// TIA Portal project "md_tarikul_islam_sheam(Batch_04)_roll_25_distribution" (V18)

(* hardware
DEVICE "S7-1500/ET200MP station_1"  S7-1500 station
   slot 0: "Rail_0"  Rack  6ES7 590-1***0-0AA0
   slot 1: "PLC_1"  CPU 1516-3 PN/DP  6ES7 516-3AN02-0AB0  V2.9
      slot 3: "CPU display_1"  6ES7591-1BA00-0AA0
      slot 32768: "PROFINET interface_1"  X1
      slot 33024: "PROFINET interface_2"  X2
      slot 33280: "DP interface_1"  X3
      slot 34817: "Virtual CP interface port_1"  Virtual CP interface port  Virtual CP interface port
   slot 2: "DI 32x24VDC HF_1"  DI 32x24VDC HF  6ES7 521-1BL00-0AB0  V2.2
   slot 3: "DQ 32x24VDC/0.5A HF_1"  DQ 32x24VDC/0.5A HF  6ES7 522-1BL01-0AB0  V1.1
   slot 4: "AI 8xU/I/RTD/TC ST_1"  AI 8xU/I/RTD/TC ST  6ES7 531-7KF00-0AB0  V2.2
   slot 5: "AQ 4xU/I ST_1"  AQ 4xU/I ST  6ES7 532-5HD00-0AB0  V2.2
DEVICE "HMI_1"  TP700 Comfort
   slot 0: "HMI_1"  TP700 Comfort  6AV2 124-0GC01-0AX0  17.0.0.0
   slot 1: "HMI_RT_1"  TP700 Comfort  6AV2 124-0GC01-0AX0  17.0.0.0
   slot 5: "HMI_1.IE_CP_1"  PROFINET Interface  17.0.0.0
      slot 1: "PROFINET Interface_1"  PROFINET Interface
         slot 1: "Port_1"  Port
         slot 2: "Port_2"  Port
   slot 7: "HMI_1.MPI/DP_CP_1"  MPI/DP Interface  17.0.0.0
*)

// ===== PLC "PLC_1"  CPU 1516-3 PN/DP =====

VAR_GLOBAL   // PLC tag table "Default tag table"
   "start" AT %I1.0 : Bool;
END_VAR

VAR_GLOBAL   // PLC tag table "Tag table_1"
   "is_mag_empty" AT %I0.6 : Bool;
   "ejecter_retracted" AT %I0.4 : Bool;
   "ejector_adv" AT %I0.5 : Bool;
   "con_fwd" AT %Q0.0 : Bool;
   "cov_back" AT %Q0.1 : Bool;
   "wp_end" AT %I0.2 : Bool;
   "stop" AT %I1.1 : Bool;
   "mag_empty_led" AT %Q1.2 : Bool;
   "advanced_slide" AT %Q0.4 : Bool;
   "cyl_advance" AT %M8.0 : Bool;
   "cyl_return" AT %M7.1 : Bool;
   "conv_fwd" AT %M7.2 : Bool;
   "cov_stop" AT %M7.3 : Bool;
   "end" AT %M7.4 : Bool;
   "mag_empty_relay" AT %M7.0 : Bool;
   "emo_relay" AT %M7.5 : Bool;
   "reset" AT %I1.3 : Bool;
   "reset_relay" AT %M7.6 : Bool;
   "mem_stop" AT %M2.0 : Bool;
   "meme_start" AT %M2.3 : Bool;
   "Tag_1" AT %M2.6 : Bool;
   "PRODUCT_END" AT %M2.7 : Bool;
   "mem_start_indicator" AT %M6.0 : Bool;
   "mem_stop_indicator" AT %M6.1 : Bool;
   "start_indicator_light" AT %Q1.0 : Bool;
   "stop_indicator_light" AT %Q1.3 : Bool;
   "reset_indicator" AT %Q1.1 : Bool;
   "mem_ready_to_go" AT %M9.0 : Bool;
   "mem_reset" AT %M3.0 : Bool;
   "mem_e_stop" AT %M3.2 : Bool;
END_VAR

ORGANIZATION_BLOCK "Main"   // OB1, LAD, ProgramCycle
TITLE = "Main Program Sweep (Cycle)"
{ S7_Optimized_Access := 'TRUE' }
VERSION : 0.1
   VAR_INPUT
      Initial_Call : Bool;   // Initial call of this OB
      Remanence : Bool;   // =True, if remanent data are available
   END_VAR
BEGIN

REGION Network 1
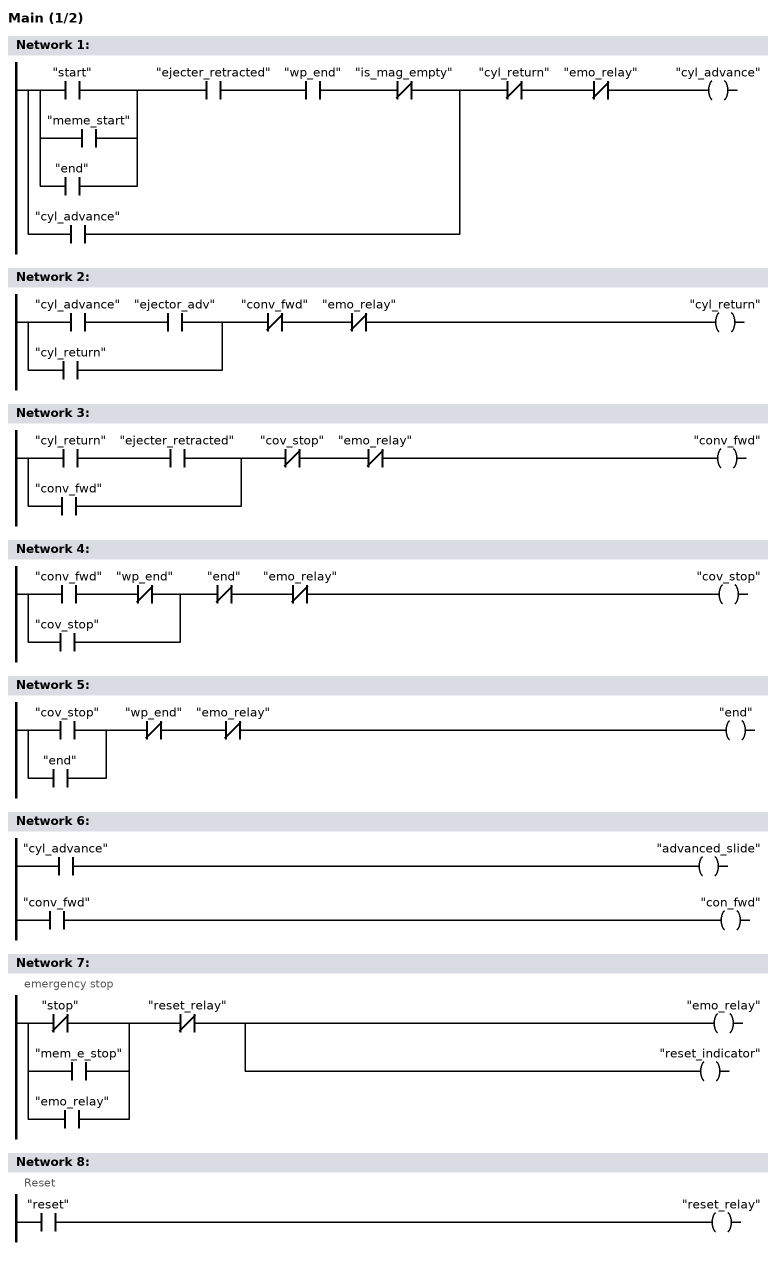
   RUNG wire#powerrail
      Contact( "start" )
      wire#w1
      Contact( "ejecter_retracted" )
      Contact( "wp_end" )
      I_Contact( "is_mag_empty" )
      wire#w2
      I_Contact( "cyl_return" )
      I_Contact( "emo_relay" )
      Coil( "cyl_advance" )
   END_RUNG
   RUNG wire#powerrail
      Contact( "meme_start" )
   END_RUNG wire#w1
   RUNG wire#powerrail
      Contact( "end" )
   END_RUNG wire#w1
   RUNG wire#powerrail
      Contact( "cyl_advance" )
   END_RUNG wire#w2
   // the same network as SCL:
   "cyl_advance" := ((("start" OR "meme_start" OR "end") AND "ejecter_retracted" AND "wp_end" AND NOT "is_mag_empty") OR "cyl_advance") AND NOT "cyl_return" AND NOT "emo_relay";
END_REGION

REGION Network 2
   RUNG wire#powerrail
      Contact( "cyl_advance" )
      Contact( "ejector_adv" )
      wire#w1
      I_Contact( "conv_fwd" )
      I_Contact( "emo_relay" )
      Coil( "cyl_return" )
   END_RUNG
   RUNG wire#powerrail
      Contact( "cyl_return" )
   END_RUNG wire#w1
   // the same network as SCL:
   "cyl_return" := (("cyl_advance" AND "ejector_adv") OR "cyl_return") AND NOT "conv_fwd" AND NOT "emo_relay";
END_REGION

REGION Network 3
   RUNG wire#powerrail
      Contact( "cyl_return" )
      Contact( "ejecter_retracted" )
      wire#w1
      I_Contact( "cov_stop" )
      I_Contact( "emo_relay" )
      Coil( "conv_fwd" )
   END_RUNG
   RUNG wire#powerrail
      Contact( "conv_fwd" )
   END_RUNG wire#w1
   // the same network as SCL:
   "conv_fwd" := (("cyl_return" AND "ejecter_retracted") OR "conv_fwd") AND NOT "cov_stop" AND NOT "emo_relay";
END_REGION

REGION Network 4
   RUNG wire#powerrail
      Contact( "conv_fwd" )
      I_Contact( "wp_end" )
      wire#w1
      I_Contact( "end" )
      I_Contact( "emo_relay" )
      Coil( "cov_stop" )
   END_RUNG
   RUNG wire#powerrail
      Contact( "cov_stop" )
   END_RUNG wire#w1
   // the same network as SCL:
   "cov_stop" := (("conv_fwd" AND NOT "wp_end") OR "cov_stop") AND NOT "end" AND NOT "emo_relay";
END_REGION

REGION Network 5
   RUNG wire#powerrail
      Contact( "cov_stop" )
      wire#w1
      I_Contact( "wp_end" )
      I_Contact( "emo_relay" )
      Coil( "end" )
   END_RUNG
   RUNG wire#powerrail
      Contact( "end" )
   END_RUNG wire#w1
   // the same network as SCL:
   "end" := ("cov_stop" OR "end") AND NOT "wp_end" AND NOT "emo_relay";
END_REGION

REGION Network 6
   RUNG wire#powerrail
      Contact( "cyl_advance" )
      Coil( "advanced_slide" )
   END_RUNG
   RUNG wire#powerrail
      Contact( "conv_fwd" )
      Coil( "con_fwd" )
   END_RUNG
   // the same network as SCL:
   "advanced_slide" := "cyl_advance";
   "con_fwd" := "conv_fwd";
END_REGION

REGION Network 7
   // emergency stop
   RUNG wire#powerrail
      I_Contact( "stop" )
      wire#w1
      I_Contact( "reset_relay" )
      wire#w2
      Coil( "emo_relay" )
   END_RUNG
   RUNG wire#powerrail
      Contact( "mem_e_stop" )
   END_RUNG wire#w1
   RUNG wire#powerrail
      Contact( "emo_relay" )
   END_RUNG wire#w1
   RUNG wire#w2
      Coil( "reset_indicator" )
   END_RUNG
   // the same network as SCL:
   "emo_relay" := (NOT "stop" OR "mem_e_stop" OR "emo_relay") AND NOT "reset_relay";
   "reset_indicator" := "emo_relay";
END_REGION

REGION Network 8
   // Reset
   RUNG wire#powerrail
      Contact( "reset" )
      Coil( "reset_relay" )
   END_RUNG
   // the same network as SCL:
   "reset_relay" := "reset";
END_REGION

REGION Network 9
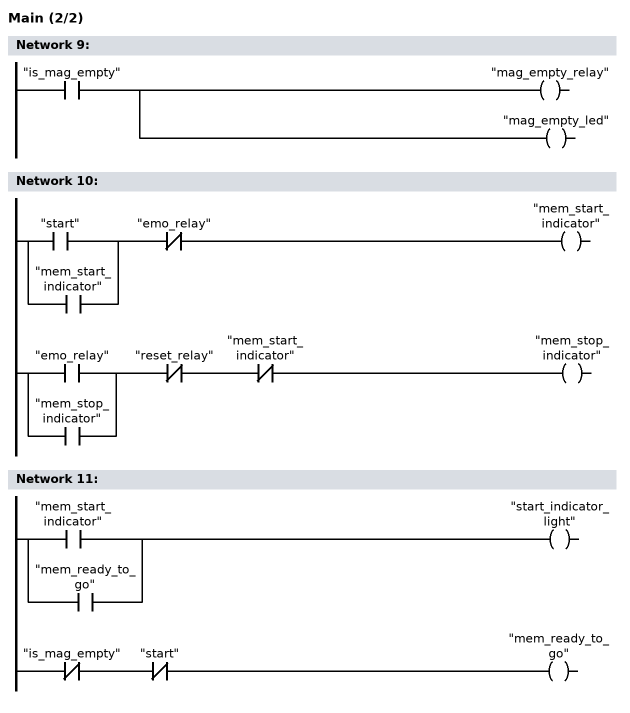
   RUNG wire#powerrail
      Contact( "is_mag_empty" )
      wire#w1
      Coil( "mag_empty_relay" )
   END_RUNG
   RUNG wire#w1
      Coil( "mag_empty_led" )
   END_RUNG
   // the same network as SCL:
   "mag_empty_relay" := "is_mag_empty";
   "mag_empty_led" := "is_mag_empty";
END_REGION

REGION Network 10
   RUNG wire#powerrail
      Contact( "start" )
      wire#w1
      I_Contact( "emo_relay" )
      Coil( "mem_start_indicator" )
   END_RUNG
   RUNG wire#powerrail
      Contact( "mem_start_indicator" )
   END_RUNG wire#w1
   RUNG wire#powerrail
      Contact( "emo_relay" )
      wire#w2
      I_Contact( "reset_relay" )
      I_Contact( "mem_start_indicator" )
      Coil( "mem_stop_indicator" )
   END_RUNG
   RUNG wire#powerrail
      Contact( "mem_stop_indicator" )
   END_RUNG wire#w2
   // the same network as SCL:
   "mem_start_indicator" := ("start" OR "mem_start_indicator") AND NOT "emo_relay";
   "mem_stop_indicator" := ("emo_relay" OR "mem_stop_indicator") AND NOT "reset_relay" AND NOT "mem_start_indicator";
END_REGION

REGION Network 11
   RUNG wire#powerrail
      Contact( "mem_start_indicator" )
      wire#w1
      Coil( "start_indicator_light" )
   END_RUNG
   RUNG wire#powerrail
      Contact( "mem_ready_to_go" )
   END_RUNG wire#w1
   RUNG wire#powerrail
      I_Contact( "is_mag_empty" )
      I_Contact( "start" )
      Coil( "mem_ready_to_go" )
   END_RUNG
   // the same network as SCL:
   "start_indicator_light" := "mem_start_indicator" OR "mem_ready_to_go";
   "mem_ready_to_go" := NOT "is_mag_empty" AND NOT "start";
END_REGION
END_ORGANIZATION_BLOCK

(* ===== HMI "HMI_RT_1" =====
system functions are stored by id; their names below are inferred from use
connection "HMI_Connection_1": ETHERNET, S7_1500_OMS

HMI tags "Default tag table"
   "meme_start" : Bool = PLC meme_start AT %M2.3, 1 s
   "mem_stop" : Bool = PLC mem_stop AT %M2.0, 1 s
   "reset_relay" : Bool = PLC reset_relay AT %M7.6, 1 s
   "mag_empty_relay" : Bool = PLC mag_empty_relay AT %M7.0, 1 s
   "r_cyl_adv" : Bool = PLC cyl_advance AT %M8.0, 1 s
   "r_cov_stop" : Bool = PLC cov_stop AT %M7.3, 1 s
   "Tag_1" : Bool = PLC Tag_1 AT %M2.6, 1 s
   "PRODUCT_END" : Bool = PLC PRODUCT_END AT %M2.7, 1 s
   "con_fwd" : Bool = PLC con_fwd AT %Q0.0, 1 s
   "r_conv_fwd" : Bool = PLC conv_fwd AT %M7.2, 1 s
   "mem_e_stop" : Bool = PLC mem_e_stop AT %M3.2, 1 s
   "mem_reset" : Bool = PLC mem_reset AT %M3.0, 1 s

screen "Root screen" 800x480, template "Template_1"
   Button "Button_1" at 362,107 size 113x53; TextOff 'START'
      on Press: function_b14e0dd5("meme_start", 0)
   Button "Button_2" at 361,179 size 114x55; TextOff 'STOP'
      on Press: function_b14e0dd5("mem_e_stop", 0)
   TextField "Text field_1" at 339,50 size 167x23; Text 'Distribution_Task'

Template "Template_1" 800x480
   Button "Exit" at 720,420 size 78x58; TextOff 'Exit'; PictureOff "ExitRuntime_TP700_Comfort_TR"; PictureOn "ExitRuntime_TP700_Comfort_TR"
      on Release: StopRuntime(0)
   Button "Template_Button" at 640,420 size 78x58; TextOff 'Text'
   Button "Template_Button_1" at 560,420 size 78x58; TextOff 'Text'
   Button "Template_Button_2" at 480,420 size 78x58; TextOff 'Text'
   Button "Template_Button_3" at 400,420 size 78x58; TextOff 'Text'
   Button "Template_Button_4" at 321,420 size 78x58; TextOff 'Text'
   Button "Template_Button_5" at 241,420 size 78x58; TextOff 'Text'
   Button "Template_Button_6" at 161,420 size 78x58; TextOff 'Text'
   Button "Template_Button_7" at 81,420 size 78x58; TextOff 'Text'
   Button "Start screen" at 1,420 size 78x58; TextOff 'Start screen'; PictureOff "NavigateHome_TP700_Comfort_TR"; PictureOn "NavigateHome_TP700_Comfort_TR"
      on Release: ActivateScreen("Root screen", 0)
*)